// TIA Portal V20 export
TYPE "LConSMC_typeTorqueValues"
// stored: Access Published
   STRUCT
      upperTorqueLimit : LReal;
      lowerTorqueLimit : LReal;
      additiveTorque : LReal;
   END_STRUCT;
END_TYPE
